TYPE DUT_HMI_10 :
STRUCT
	Manuals : DUT_HMI_10_MANUALS;
	ProductStatus 	: eProductStatus;
	State			: eStationState;
	EVDiagnostic 	: ARRAY[0..20] OF DUT_HMI_EV_Diagnostic;
	EVInfo			: ARRAY[0..CNC.NUM_MAX_MANUALS_10-1] OF DUT_HMI_EV_Info;
	Status			: USINT;
	CycleTime		: STRING;
	BroachTarget	: USINT;
END_STRUCT
END_TYPE

(* stored: Version 1.1.0.1, ProductVersion 3.1.4024.15
   DUT DUT_HMI_10: Id {0643d7a1-1de8-4775-b394-fafdae9efe4b} *)
